{attribute 'qualified_only'}
{attribute 'strict'}
{attribute 'to_string'}
TYPE eForceBool:
(
	none := 0,
	On	:= 1,
	Off := 2
);
END_TYPE

(* stored: Version 1.1.0.1, ProductVersion 3.1.4026.18
   DUT eForceBool: Id {2c25cd44-78fc-41f3-aae3-58dc2bc7cd22} *)
